PROGRAM PG_Calculate_Sun
VAR
	Sun_history: FB_DataHistory_Int;
	INT_TRIG_0: INT_TRIG;
	FB_Sonne_1: FB_Sonne;
	R_TRIG_0: R_TRIG;
END_VAR
VAR // added by the converter: edge detectors and wires of the graphical bodies
    _w1 : BOOL;
END_VAR

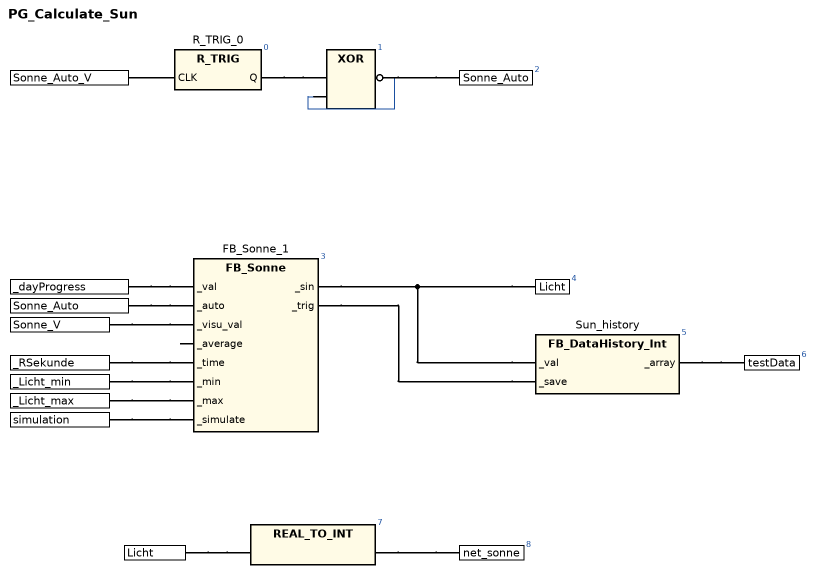
R_TRIG_0(CLK := Sonne_Auto_V); // R_TRIG
_w1 := R_TRIG_0.Q XOR NOT _w1;
Sonne_Auto := NOT _w1;
FB_Sonne_1(
    _val := _dayProgress,
    _auto := Sonne_Auto,
    _visu_val := Sonne_V,
    _time := _RSekunde,
    _min := _Licht_min,
    _max := _Licht_max,
    _simulate := simulation); // FB_Sonne
Licht := FB_Sonne_1._sin;
Sun_history(_val := FB_Sonne_1._sin, _save := FB_Sonne_1._trig); // FB_DataHistory_Int
testData := Sun_history._array;
net_sonne := REAL_TO_INT(Licht);

END_PROGRAM

(* stored: Version 1.1.0.1, ProductVersion 3.1.4018.5
   POU PG_Calculate_Sun: Id {6f2d8c91-1a48-4e18-a6d3-ae78ffda30c8}, SpecialFunc None *)
